// TIA Portal V19 export
TYPE "LEXCHANGETRAY_typeSr1000ProfinetTelegram_matchingLevelandTotalEvaluationGradeStatus"
// stored: Access Published
   STRUCT
      statusBytes : Array[0..5] of Byte;
      matchingLevel : UInt;
      isoIec15415 : UInt;
      aimdpmGrade : UInt;
   END_STRUCT;
END_TYPE
